// TIA Portal V15 SP1 export
// export: Created 2018-01-22T18:38:18.8737467Z, ExportSetting WithDefaults, DisplayName Totally Integrated Automation Portal, DisplayVersion V15 SP1, DisplayName TIA Portal Openness, DisplayVersion V15 SP1, DisplayName TIA Portal Version Control Interface, DisplayVersion V15 SP1, DisplayName Development Version TIA Portal, DisplayVersion V15 SP1, DisplayName STEP 7 Professional, DisplayVersion V15 SP1, DisplayName SIMATIC Energy Suite, DisplayVersion V15 SP1, DisplayName WinCC Professional, DisplayVersion V15 SP1
FUNCTION "Block_3" : Void   // FC1, LAD
{ S7_Optimized_Access := 'TRUE' }
VERSION : 0.1
// stored: AutoNumber true, IsIECCheckEnabled false, SetENOAutomatically False, UDAEnableTagReadback false
BEGIN
END_FUNCTION
